// TIA Portal project "训练一学习DB" (V16)

(* hardware
DEVICE "S7-1200 station_1"  S7-1200 Station
   slot 0: "Rack_0"  S7-1200 Rack  Rack  V1.0
   slot 1: "PLC_1"  CPU 1214C DC/DC/DC  6ES7 214-1AG40-0XB0  V4.4
*)

// ===== PLC "PLC_1"  CPU 1214C DC/DC/DC =====

DATA_BLOCK "队列数据"   // DB1
{ S7_Optimized_Access := 'FALSE' }
VERSION : 0.1
   VAR
      随机生成数据 : Bool;
      上一个周期1 : Bool;
      数据 : DTL;
      RLV : Int;
      中间变量1 : UDInt;
      加入队列 : Bool;
      上一个周期2 : Bool;
      队列 : Array[0..9] of UDInt;
      inter : DInt;
      踢出队列 : Bool;
      上一个周期3 : Bool;
      踢出队列中间转换数组 : Array[0..9] of UDInt;
      inter2 : UDInt;
   END_VAR
BEGIN
END_DATA_BLOCK

FUNCTION "MHJ-PLC-Lab-Function-S71200" : Void   // FC9000, SCL
{ S7_Optimized_Access := 'TRUE' }
VERSION : 0.1
   VAR_TEMP
      rdTimeReturn : Int;
      outputTime : DTL;
      SyncVal : Byte;
      forVal : Int;
      forVal_2 : Int;
      Value : Byte;
   END_VAR
   VAR CONSTANT
      CompVal : Byte := 16#34;
      Value_01 : Byte := 16#11;
      Value_01_DW : DWord := 16#A165_D992;
      Value_02_DW : DWord := 16#58BE_4401;
   END_VAR
BEGIN

   #Value:=PEEK(area := 16#82,
        dbNumber := 0,
        byteOffset := 511);
   #Value := #Value + 1;

   POKE(area := 16#82,
        dbNumber := 0,
        byteOffset := 511,
        value := #Value);

   POKE(area:=16#81,
        dbNumber:=0,
        byteOffset:=1016,
        value:=#Value_01_DW);
   POKE(area := 16#81,
        dbNumber := 0,
        byteOffset := 1020,
        value := #Value_02_DW);

   POKE(area := 16#81,
        dbNumber := 0,
        byteOffset := 511,
        value := B#16#00);

   FOR #forVal := 0 TO 120 DO
       FOR #forVal_2:=0 TO 10 DO
           #rdTimeReturn:=RD_SYS_T(#outputTime);
           #rdTimeReturn := WR_SYS_T(#outputTime);
           #rdTimeReturn := RD_SYS_T(#outputTime);
           #rdTimeReturn := WR_SYS_T(#outputTime);
       END_FOR;
       #SyncVal:= PEEK(area := 16#81,
                      dbNumber := 0,
                      byteOffset := 511);
       IF #SyncVal = #CompVal THEN
          GOTO M_1;
       END_IF;
   END_FOR;
   RETURN;

   M_1:
   POKE(area := 16#81,
        dbNumber := 0,
        byteOffset := 511,
        value := B#16#0);
END_FUNCTION

ORGANIZATION_BLOCK "Main"   // OB1, LAD, ProgramCycle
TITLE = "Main Program Sweep (Cycle)"
{ S7_Optimized_Access := 'TRUE' }
VERSION : 0.1
   VAR_INPUT
      Initial_Call : Bool;   // Initial call of this OB
      Remanence : Bool;   // =True, if remanent data are available
   END_VAR
   VAR_TEMP   // added for the SCL form of the ladder/FBD networks
      _w1 : Bool;
   END_VAR
BEGIN

REGION Network 1: 随机生成一个数据
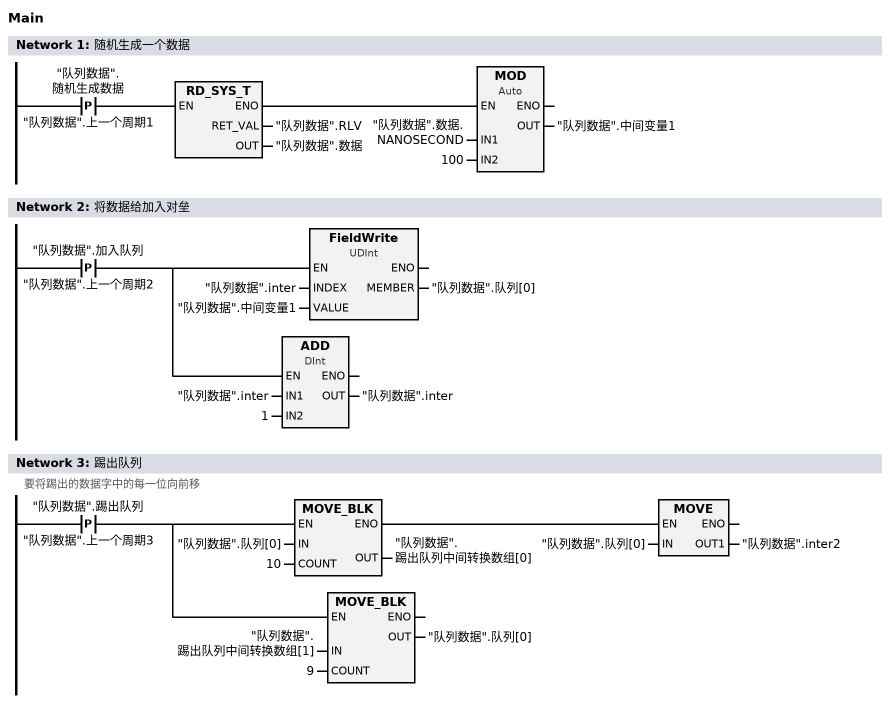
   // ENO of a box is taken as its EN; it also drops when the box reports an error
   #_w1 := "队列数据".随机生成数据 AND NOT "队列数据".上一个周期1;   // rising edge of "队列数据".随机生成数据
   "队列数据".上一个周期1 := "队列数据".随机生成数据;
   IF #_w1 THEN
       "队列数据".RLV := RD_SYS_T(OUT => "队列数据".数据);
       "队列数据".中间变量1 := "队列数据".数据.NANOSECOND MOD 100;
   END_IF;
END_REGION

REGION Network 2: 将数据给加入对垒
   // no SCL statement known for FieldWrite: written as a call
   #_w1 := "队列数据".加入队列 AND NOT "队列数据".上一个周期2;   // rising edge of "队列数据".加入队列
   "队列数据".上一个周期2 := "队列数据".加入队列;
   IF #_w1 THEN
       FieldWrite(index := "队列数据".inter, value := "队列数据".中间变量1, member => "队列数据".队列[0]);
       "队列数据".inter := "队列数据".inter + 1;
   END_IF;
END_REGION

REGION Network 3: 踢出队列
   // 要将踢出的数据字中的每一位向前移
   #_w1 := "队列数据".踢出队列 AND NOT "队列数据".上一个周期3;   // rising edge of "队列数据".踢出队列
   "队列数据".上一个周期3 := "队列数据".踢出队列;
   IF #_w1 THEN
       MOVE_BLK(IN := "队列数据".队列[0], COUNT := 10, OUT => "队列数据".踢出队列中间转换数组[0]);
       "队列数据".inter2 := "队列数据".队列[0];
       MOVE_BLK(IN := "队列数据".踢出队列中间转换数组[1], COUNT := 9, OUT => "队列数据".队列[0]);
   END_IF;
END_REGION
END_ORGANIZATION_BLOCK